TYPE ST_DB_Solvents :
STRUCT
	solvent_ID   : DINT;

    solventName1 : STRING(80);
    density1     : STRING(40);

    addedBy      : STRING(80);
    addedDate    : STRING(40);

    solventName2 : STRING(80);
    solventName3 : STRING(80);
    solventName4 : STRING(80);

    density2     : STRING(40);
    density3     : STRING(40);
    density4     : STRING(40);
END_STRUCT
END_TYPE

(* stored: Version 1.1.0.1, ProductVersion 3.1.4024.15
   DUT ST_DB_Solvents: Id {1bfa9040-df66-4d57-bc6b-8fbfa8b0d911} *)
